(* Schneider Machine Expert - Basic project State1_TestingwithATV320, file version 2.7.0.0 *)
(* ProjectInformations: Name=New project *)

HARDWARE
  Cpu 0: TM221ME16T/G
  ModuleExtensionObject 0: TM3AM6/G
  EthernetConfiguration: NetworkName=M221, IpAllocationMode=FixedAddress, IpAddress=192.168.3.84, SubnetMask=255.255.255.0
  SerialLineConfiguration: Baud=Baud19200, Parity=ParityEven, DataBits=DataBits8, StopBits=StopBits1, PhysicalMedium=PhysicalMediumRs485, TransmissionMode=TransmissionModeModbusRtu, SlaveId=1, Addressing=MasterAddressing
  MastTask: UsePeriodScanMode=false, PeriodScan=100
  FastTask: Period=255
  CpuBehavior: StartingMode=StartAsPreviousState, AutoSaveRamOnEeprom=true, WatchdogPeriod=250

SYMBOLS  (address, symbol, comment, settings)
  %MW0      MW_SLOT1_AO_CH0_SP
  %MF0      FLOAT_SETPOINT0
  %MC_POWER_ATV0 A1  [Axis(Value(DriveAxis=None))]
  %I0.0     I_CH0_SW_FWD
  %I0.1     I_CH1_SW_BWD
  %Q0.0     O_CH0_FW_CMD
  %Q0.1     O_CH1_BW_CMD
  %IW1.0    SLOT1_AI_CHANNEL0  [Type=Type_0_10V, Scope=Scope_Customized, Minimum=0, Maximum=10000]
  %IW1.1    SLOT1_AI_CHANNEL1  [Type=Type_0_10V, Scope=Scope_Customized, Minimum=0, Maximum=10000]
  %IW1.2    SLOT1_AI_CHANNEL2  [Type=Type_0_10V, Scope=Scope_Customized, Minimum=0, Maximum=10000]
  %IW1.3    SLOT1_AI_CHANNEL3  [Type=Type_0_10V, Scope=Scope_Customized, Minimum=0, Maximum=10000]
  %QW1.0    SLOT1_AO_CHANNEL0  [Type=Type_0_10V, Scope=Scope_Customized, Minimum=0, Maximum=10000]
  %QW1.1    SLOT1_AO_CHANNEL1  [Type=Type_0_10V, Scope=Scope_Customized, Minimum=0, Maximum=10000]

POU New POU
  (* SectionNumber=1 *)

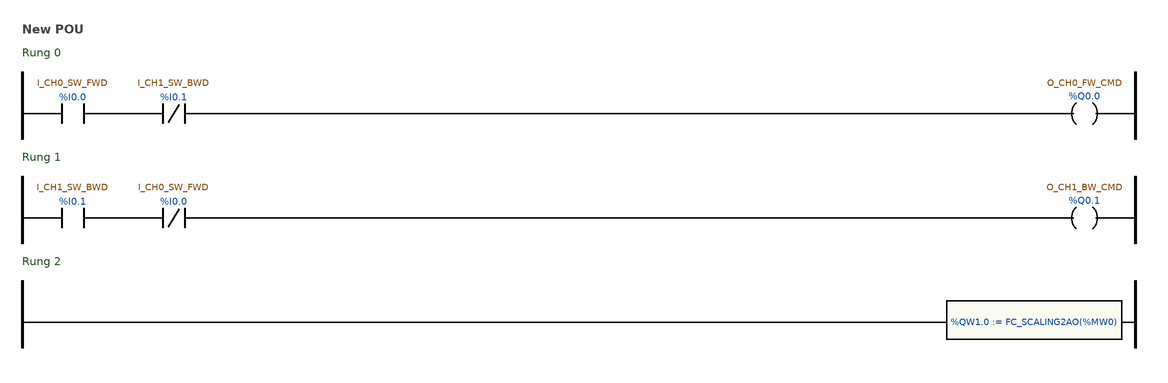

// Rung 0
  LD %I0.0                (* I_CH0_SW_FWD *)
  ANDN %I0.1              (* I_CH1_SW_BWD *)
  ST %Q0.0                (* O_CH0_FW_CMD *)
  // as ST:
  //   O_CH0_FW_CMD := I_CH0_SW_FWD AND NOT I_CH1_SW_BWD;

// Rung 1
  LD %I0.1                (* I_CH1_SW_BWD *)
  ANDN %I0.0              (* I_CH0_SW_FWD *)
  ST %Q0.1                (* O_CH1_BW_CMD *)
  // as ST:
  //   O_CH1_BW_CMD := I_CH1_SW_BWD AND NOT I_CH0_SW_FWD;

// Rung 2
  LD 1
  [ %QW1.0 := FC_SCALING2AO ( %MW0 ) ](* SLOT1_AO_CHANNEL0, MW_SLOT1_AO_CH0_SP *)
  // as ST:
  //   SLOT1_AO_CHANNEL0 := FC_SCALING2AO ( MW_SLOT1_AO_CH0_SP );

UserFunctionPou FC_SCALING2AO
  (* SectionNumber=2 *)

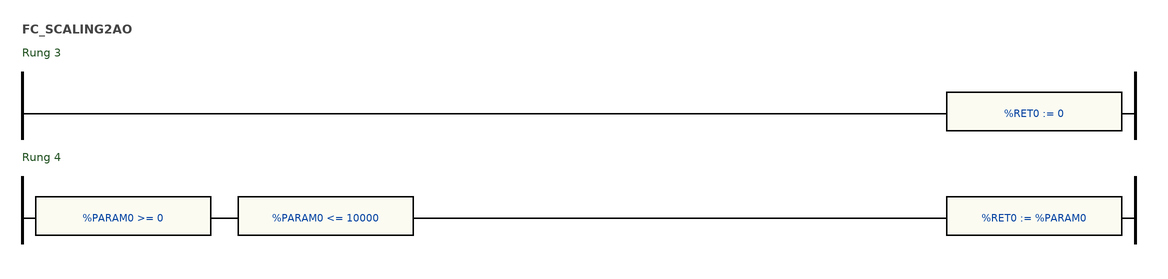

// Rung 3
  LD 1
  [ %RET0 := 0 ]
  // as ST:
  //   %RET0 := 0;

// Rung 4
  LD [ %PARAM0 >= 0 ]
  AND [ %PARAM0 <= 10000 ]
  [ %RET0 := %PARAM0 ]
  // as ST:
  //   IF %PARAM0 >= 0 AND %PARAM0 <= 10000 THEN %RET0 := %PARAM0; END_IF;
